# EPICS autosave request: ipApp/Db/Oxford_CS800.req
$(P)$(Q):RRATE
$(P)$(Q):RTEMP
$(P)$(Q):PTIME
$(P)$(Q):CTEMP
$(P)$(Q):ERATE
$(P)$(Q):DISABLE
